FUNCTION_BLOCK F_GE_3 (* greater or equal (3 inputs) *)
  (* Standard: 61131-3; Classification: standard comparison function; Description: Copyright (c) 2011 TU Wien ACIN and others. This program and the accompanying materials are made available under the terms of the Eclipse Public License 2.0 which is available at https://www.eclipse.org/legal/epl-2.0/ SPDX-License-Identifier: EPL-2.0 Some portions generated by Gemini CLI *)
  (* Version 1.0, 2026-01-31, Franz Höpfinger, HR Agrartechnik GmbH, conform to IEC 61131-3, copy F_GE and make this. *)
  PACKAGE iec61131::comparison;
  {SET_ATTRIBUTE(eclipse4diac::core::GenericClassName, 'GEN_GE')}
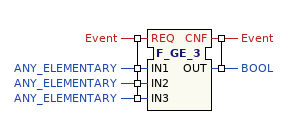
  EVENT_INPUT
    REQ WITH IN1, IN2, IN3; (* Service Request *)
  END_EVENT
  EVENT_OUTPUT
    CNF WITH OUT; (* Confirmation of Requested Service *)
  END_EVENT
  VAR_INPUT
    IN1 : ANY_ELEMENTARY; (* Input value 1 *)
    IN2 : ANY_ELEMENTARY; (* Input value 2 *)
    IN3 : ANY_ELEMENTARY; (* Input value 3 *)
  END_VAR
  VAR_OUTPUT
    OUT : BOOL; (* value 1 >= value2 >= value3 => true *)
  END_VAR
END_FUNCTION_BLOCK
